FUNCTION_BLOCK FB_Optiflux5000_EL3022 IMPLEMENTS I_VolumeFlowSensor
VAR_INPUT
END_VAR
VAR_OUTPUT
END_VAR
VAR								
	//Property Real value
	fVolFlow : REAL;
	//Raw value
	VolFlowRaw AT %I* : INT;
	//Convertion parameters
	m : REAL := 0.1098666341; //Multiplier for convertion
END_VAR

// Volume Flow measurement with Krohne Optiflux 5000
// https://www.krohne.com/de-de/produkte/durchflussmesstechnik/komponenten-und-zusaetzliche-betriebsmittel-fuer-die-durchflussmessung/messwertaufnehmer/optiflux-5000

PROPERTY VolumeFlow : REAL
GET
fVolFlow := m * INT_TO_REAL(VolFlowRaw);
VolumeFlow := THIS^.fVolFlow;
END_GET
END_PROPERTY

END_FUNCTION_BLOCK

(* stored: Version 1.1.0.1
   POU FB_Optiflux5000_EL3022: Id {993a7f08-d4e9-4a4b-81b1-d13df2987775}, SpecialFunc None
   Property VolumeFlow: Id {a8f81ea5-c692-4837-9874-9e77a19b3686}
   Get Get: Id {d0be21c8-fd5c-4567-ae96-7ea0a2f352bf} *)
